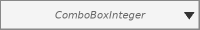
VISUALIZATION VISU_HELPER_Combobox_eReglertyp  // 200x30
VAR_IN_OUT
    varEnum : eReglertyp;
END_VAR
    ComboBoxInteger (0,0 200x30), variable: varEnum, text list: 'TextListForCombobox_eReglertyp'
END_VISUALIZATION

(* stored: Version 1.1.0.1, ProductVersion 3.1.4024.12
   Visu VISU_HELPER_Combobox_eReglertyp: Id {5526bff5-3237-471a-a656-174b78cc3102} *)
